{attribute 'qualified_only'}
{attribute 'strict'}
{attribute 'to_string'}
TYPE eLiftposition :
(
	Home 		:= 0,
	Position_1	:= 1,
	Position_2	:= 2,
	Position_3	:= 3,
	Position_4	:= 4,
	Position_5	:= 5,
	GoingUp 	:= 6,
	GoingDown 	:= 7
	
);
END_TYPE

(* stored: Version 1.1.0.1
   DUT eLiftposition: Id {8e6f9247-8a73-46d2-b330-6ef24caf6819} *)
